// TIA Portal V20 export
VAR_GLOBAL   // PLC tag table "IO_PLC_Centralizer_PLC_Functional_Test_Rework"
   In AT %I600.0 : "IO_Device_Functinal_Test_Rework";
   Out AT %Q600.0 : "IO_Device_Test_Parameters_Rework";
END_VAR
